FUNCTION TryConvert_SINT_TO_UDINT : BOOL
VAR_INPUT
	in : SINT;
	out : REFERENCE TO UDINT;
END_VAR

IF in < DatatypeLimits.MIN_VALUE_OF_SINT_WHICH_CAN_BE_HELD_IN_A_UDINT THEN
	RETURN;
END_IF

out := SINT_TO_UDINT(in);
TryConvert_SINT_TO_UDINT := TRUE;

END_FUNCTION

(* stored: Version 1.1.0.1, ProductVersion 3.1.4024.12
   POU TryConvert_SINT_TO_UDINT: Id {104228fa-7132-40b6-91ee-843fed613391}, SpecialFunc None *)
